{attribute 'strict'}
TYPE E_ASDAB3_State :
(
	ASDAB3_UNINITIALIZED := 0,
	ASDAB3_INITIALIZING	:= 10,
	ASDAB3_READY_INITIALIZED := 20,
	ASDAB3_IDLE	:= 25,
	ASDAB3_MOVE_ABSOLUTE := 30,
	ASDAB3_MOVE_ABSOLUTE_DONE := 40,
	ASDAB3_HOME := 50,
	ASDAB3_HOME_DONE := 60,
	ASDAB3_RESET := 70,
	ASDAB3_RESET_DONE := 80,
	ASDAB3_ABORTING := -10
	
);
END_TYPE

(* stored: Version 1.1.0.1, ProductVersion 3.1.4024.12
   DUT E_ASDAB3_State: Id {990f3738-9a57-4e5e-b036-f32692d7bab0} *)
